FUNCTION_BLOCK CAMERA (* Camera OpenCV function block *)
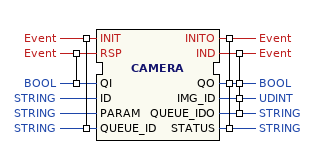
  EVENT_INPUT
    INIT WITH , DEVICE_ID, QUEUE_ID;
    RSP WITH QI;
  END_EVENT
  EVENT_OUTPUT
    INITO WITH QO, STATUS;
    IND WITH QO, IMG_ID, QUEUE_IDO, STATUSO;
  END_EVENT
  VAR_INPUT
    QI : BOOL;
    ID : STRING;
    PARAM : STRING;
    QUEUE_ID : STRING;
  END_VAR
  VAR_OUTPUT
    QO : BOOL;
    IMG_ID : UDINT;
    QUEUE_IDO : STRING;
    STATUS : STRING;
  END_VAR
END_FUNCTION_BLOCK
